// TIA Portal V18 export
DATA_BLOCK "L1_prgTaglio"   // DB25
{ S7_Optimized_Access := 'TRUE' }
VERSION : 0.1
// stored: AutoNumber false, DBAccessibleFromOPCUA true, DBAccessibleFromWebserver true, IsOnlyStoredInLoadMemory false, IsRetainMemResEnabled false, IsWriteProtectedInAS false, MemoryReserve 0
   VAR RETAIN
      data : "LGasp_Tagliosega";
   END_VAR
BEGIN
END_DATA_BLOCK
